FUNCTION_BLOCK EmergencySludgeBuffer_HMI (* Service Interface Function Block Type *)
  (* Standard: 61499-2 *)
  (* Version 0.0, 7/4/2026, Schneider Electric, template *)
  PACKAGE SE.Nereda;
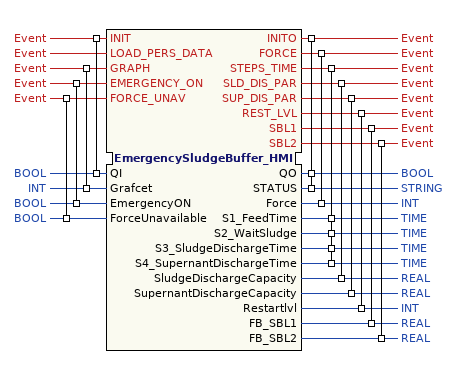
  EVENT_INPUT
    INIT WITH QI;
    LOAD_PERS_DATA;
    GRAPH WITH Grafcet;
    EMERGENCY_ON WITH EmergencyON;
    FORCE_UNAV WITH ForceUnavailable;
  END_EVENT
  EVENT_OUTPUT
    INITO WITH QO, STATUS;
    FORCE WITH Force;
    STEPS_TIME WITH S1_FeedTime, S2_WaitSludge, S3_SludgeDischargeTime, S4_SupernantDischargeTime;
    SLD_DIS_PAR WITH SludgeDischargeCapacity;
    SUP_DIS_PAR WITH SupernantDischargeCapacity;
    REST_LVL WITH Restartlvl;
    SBL1 WITH FB_SBL1;
    SBL2 WITH FB_SBL2;
  END_EVENT
  VAR_INPUT
    QI : BOOL;
    Grafcet : INT;
    EmergencyON : BOOL;
    ForceUnavailable : BOOL;
  END_VAR
  VAR_OUTPUT
    QO : BOOL; (* Event Output Qualifier *)
    STATUS : STRING; (* Service Status *)
    Force : INT;
    S1_FeedTime : TIME;
    S2_WaitSludge : TIME;
    S3_SludgeDischargeTime : TIME;
    S4_SupernantDischargeTime : TIME;
    SludgeDischargeCapacity : REAL;
    SupernantDischargeCapacity : REAL;
    Restartlvl : INT;
    FB_SBL1 : REAL;
    FB_SBL2 : REAL;
  END_VAR
  SERVICE /
    SEQUENCE 
    END_SEQUENCE
  END_SERVICE
END_FUNCTION_BLOCK
